SUBAPPLICATION AX_OR_AND_3_SPLIT (* 3 unabhaengige AX-Signale je einzeln durchreichen (OUT1/OUT2/OUT3 = IN1/IN2/IN3) sowie gemeinsam UND- (OUT_AND/OUT_AND2 = IN1 AND IN2 AND IN3) und ODER-verknuepfen (OUT_OR/OUT_OR2 = IN1 OR IN2 OR IN3). *)
  (* Standard: 61499-2 *)
  (* Version 1.0, 2026-09-17, Franz Höpfinger, Meisterschulen am Ostbahnhof, Erweitert um UND- und ODER-Sammelverknuepfungen (OUT_AND/OUT_AND2, OUT_OR/OUT_OR2) mit aufgedoppelten Ausgangszweigen (AX_SPLIT_2) und bereinigten FB-Instanznamen. *)
  PACKAGE MyLib::sys;
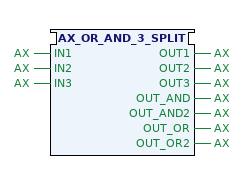
  SOCKETS
    IN1 : adapter::types::unidirectional::AX; (* Eingangssignal 1 *)
    IN2 : adapter::types::unidirectional::AX; (* Eingangssignal 2 *)
    IN3 : adapter::types::unidirectional::AX; (* Eingangssignal 3 *)
  END_SOCKETS
  PLUGS
    OUT1 : adapter::types::unidirectional::AX; (* Durchgereichtes Eingangssignal 1 (IN1) *)
    OUT2 : adapter::types::unidirectional::AX; (* Durchgereichtes Eingangssignal 2 (IN2) *)
    OUT3 : adapter::types::unidirectional::AX; (* Durchgereichtes Eingangssignal 3 (IN3) *)
    OUT_AND : adapter::types::unidirectional::AX; (* IN1 AND IN2 AND IN3 - Sammelstatus alle aktiv (Zweig 1) *)
    OUT_AND2 : adapter::types::unidirectional::AX; (* IN1 AND IN2 AND IN3 - Sammelstatus alle aktiv (Zweig 2) *)
    OUT_OR : adapter::types::unidirectional::AX; (* IN1 OR IN2 OR IN3 - Sammelstatus mindestens einer aktiv (Zweig 1) *)
    OUT_OR2 : adapter::types::unidirectional::AX; (* IN1 OR IN2 OR IN3 - Sammelstatus mindestens einer aktiv (Zweig 2) *)
  END_PLUGS
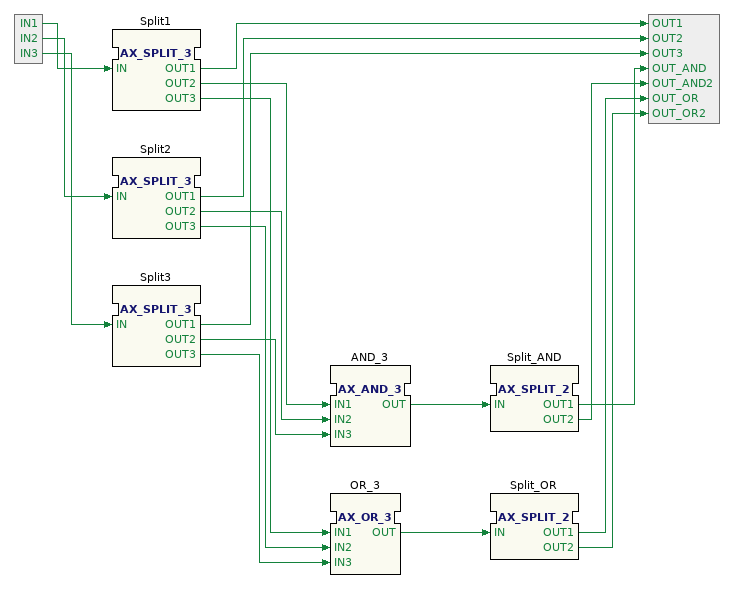
  FBS
    Split1 : adapter::events::unidirectional::AX_SPLIT_3;
    Split2 : adapter::events::unidirectional::AX_SPLIT_3;
    Split3 : adapter::events::unidirectional::AX_SPLIT_3;
    AND_3 : adapter::booleanOperators::AX_AND_3;
    Split_AND : adapter::events::unidirectional::AX_SPLIT_2;
    OR_3 : adapter::booleanOperators::AX_OR_3;
    Split_OR : adapter::events::unidirectional::AX_SPLIT_2;
  END_FBS
  ADAPTER_CONNECTIONS
    IN1 TO Split1.IN;
    IN2 TO Split2.IN;
    IN3 TO Split3.IN;
    Split1.OUT1 TO OUT1;
    Split2.OUT1 TO OUT2;
    Split3.OUT1 TO OUT3;
    Split1.OUT2 TO AND_3.IN1;
    Split2.OUT2 TO AND_3.IN2;
    Split3.OUT2 TO AND_3.IN3;
    Split1.OUT3 TO OR_3.IN1;
    Split2.OUT3 TO OR_3.IN2;
    Split3.OUT3 TO OR_3.IN3;
    AND_3.OUT TO Split_AND.IN;
    Split_AND.OUT1 TO OUT_AND;
    Split_AND.OUT2 TO OUT_AND2;
    OR_3.OUT TO Split_OR.IN;
    Split_OR.OUT1 TO OUT_OR;
    Split_OR.OUT2 TO OUT_OR2;
  END_CONNECTIONS
END_SUBAPPLICATION
